(* CODESYS project Johnson, Joachim, inlämningsuppgift Version 2.project

Project tree, tasks and I/O mapping:
  Device : CODESYS Control Win V3 x64, 3S - Smart Software Solutions GmbH, version 3.5.16.40
    application Application
      libraries: Standard, * (System)
      task MainTask (cyclic, interval t#20ms, priority 1) calls PLC_PRG
      program PLC_PRG [LD]
      global variables GVL
      Symbols
*)

// Device/Application/GVL
{attribute 'qualified_only'}
VAR_GLOBAL
	PushButton: BOOL;
	SensorOpen: BOOL;
	SensorClose: BOOL;
	MotorForward: BOOL;
	MotorReverse: BOOL;
	TopLight: BOOL;
END_VAR

// Device/Application/PLC_PRG
PROGRAM PLC_PRG
VAR
	TimmerOff: TOF; 		// Stänger av lampan efter utsatt tid på tidinsignalen.
	TimmerOn: TON; 			// Sätter på lampan efter utsatt tid på tidsinalen.
	Timmer_Elipse_Open_Door: TIME;
	Timmer_MovingDoor_On: TIME;
	Timmer_MovingDoor_off: TIME;
	
	// kanal 1. Håller koll på motorforward / stänger porten med ett par kollar mot om dörren är öppen eller ej och om motorn inte redan öppnar sig
	// kanal 2. Motsvarande kanal 1 fast öppna porten.
	// kanal 3. Hantering av lampa och blinkande lampa.
	// Får signal om någon av motorerna rör sig och har 2 timers som antingen sätter på signalen eller eller håller den avstängd
	// om dörren är öppen få den en signal från ett sidospår som håller igång lampan i 5 sekunder.
	
	LampTimmerOff: TOF; 	// The time elipse since lamp is turn off
	LampTimmerOn: TON; 		// The time elipse since lamp is turn on
	HoldDorrOpenTimer: TON; // Keeps the door open when reach the top
	DoorOpenLight: BOOL;	// Put signal to the light then the door is open.
END_VAR
VAR // added by the converter: edge detectors and wires of the graphical bodies
    _w1 : BOOL;
END_VAR

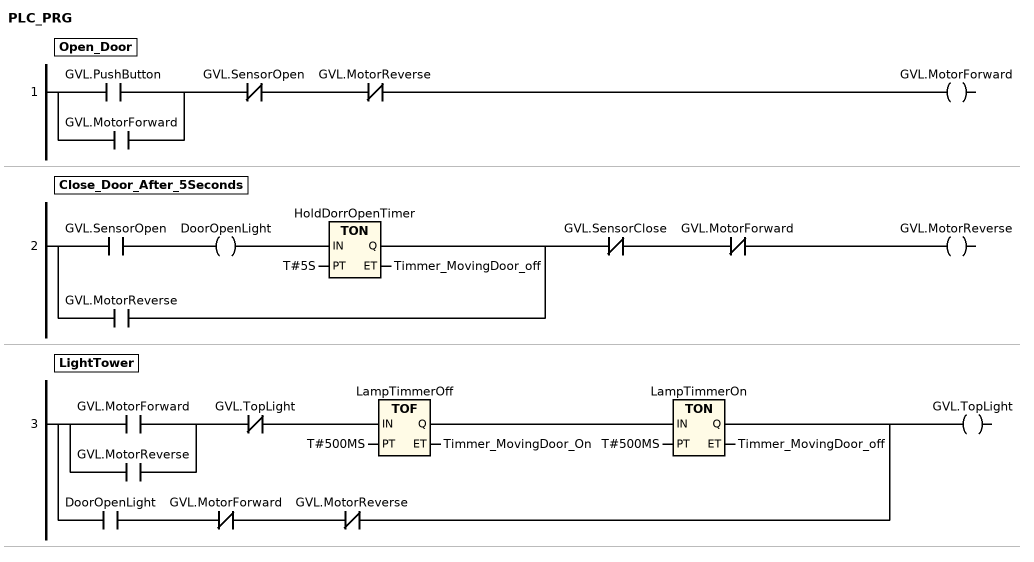
// NETWORK 1
Open_Door:
GVL.MotorForward := (GVL.PushButton OR GVL.MotorForward) AND NOT GVL.SensorOpen AND NOT GVL.MotorReverse;

// NETWORK 2
Close_Door_After_5Seconds:
DoorOpenLight := GVL.SensorOpen;
HoldDorrOpenTimer(IN := GVL.SensorOpen, PT := T#5S, ET => Timmer_MovingDoor_off); // TON
GVL.MotorReverse := (HoldDorrOpenTimer.Q OR GVL.MotorReverse) AND NOT GVL.SensorClose AND NOT GVL.MotorForward;

// NETWORK 3
LightTower:
_w1 := DoorOpenLight AND NOT GVL.MotorForward AND NOT GVL.MotorReverse;
IF NOT _w1 THEN
    LampTimmerOff(
        IN := (GVL.MotorForward OR GVL.MotorReverse) AND NOT GVL.TopLight,
        PT := T#500MS,
        ET => Timmer_MovingDoor_On); // TOF
    LampTimmerOn(IN := LampTimmerOff.Q, PT := T#500MS, ET => Timmer_MovingDoor_off); // TON
    _w1 := LampTimmerOn.Q;
END_IF
GVL.TopLight := _w1;

END_PROGRAM
